// TIA Portal V21 export
DATA_BLOCK "TimerAlarm"   // DB185
{ S7_Optimized_Access := 'FALSE' }
// stored: AutoNumber false
   VAR
      ControlKeyOff : IEC_TIMER;
      EmergencyStopPressed : IEC_TIMER;
      PowerReset : IEC_TIMER;
      CompresseDairPressurelow : IEC_TIMER;
      PowerFailure : IEC_TIMER;
      PlcRestarted : IEC_TIMER;
      Mm01FeedbackTrip : IEC_TIMER;
      Cp01FeedbackTrip : IEC_TIMER;
      Mm01OverloadTrip : IEC_TIMER;
      Cp01OverloadTrip : IEC_TIMER;
      MinimumWeightRequiredToStartmm01 : IEC_TIMER;
      Ticr01WireBreak : IEC_TIMER;
      Ticr02WireBreak : IEC_TIMER;
      Ticr03WireBreak : IEC_TIMER;
      Ticr04WireBreak : IEC_TIMER;
      Ticr05WireBreak : IEC_TIMER;
      Ticr06WireBreak : IEC_TIMER;
      Ticr07WireBreak : IEC_TIMER;
      Ticr08WireBreak : IEC_TIMER;
      Ticr09WireBreak : IEC_TIMER;
      Ticr10WireBreak : IEC_TIMER;
      Picr01WireBreak : IEC_TIMER;
      Picr02WireBreak : IEC_TIMER;
      Picr03WireBreak : IEC_TIMER;
      Picr04WireBreak : IEC_TIMER;
      Cicr01WireBreak : IEC_TIMER;
      Lc01CommunicationFailed : IEC_TIMER;
      VesselHighPressure : IEC_TIMER;
      Mm01SpeedSensorTrip : IEC_TIMER;
      PlcToHmiCommunicationFailed : IEC_TIMER;
      CipCycleOver : IEC_TIMER;
      CipCycleConductivityReached : IEC_TIMER;
      CipCycleConductivityNotReached : IEC_TIMER;
      ConductivityNotSampled : IEC_TIMER;
      CipReportDataNotLogged : IEC_TIMER;
      PhtFailed : IEC_TIMER;
      PhtPass : IEC_TIMER;
      PhtOver : IEC_TIMER;
      PhtReportDataNotLogged : IEC_TIMER;
      SterilizationTimeOver : IEC_TIMER;
      SteamFlowLow : IEC_TIMER;
      SterilizationHighTemperature : IEC_TIMER;
      SterilizationCycleCompleted : IEC_TIMER;
      SterilizationReportDataNotLogged : IEC_TIMER;
      WfiFlowLow : IEC_TIMER;
      BatchReportDataNotLogged : IEC_TIMER;
      LifeBitAlarm { S7_SetPoint := 'True'} : IEC_TIMER;
      AlarmAck_Reset { S7_SetPoint := 'True'} : IEC_TIMER;
      MasterReset { S7_SetPoint := 'True'} : IEC_TIMER;
   END_VAR
BEGIN
END_DATA_BLOCK
